{attribute 'GeneratedUsingTerminal: EL3201-0030-0022'}
{attribute addProperty BoxType "EL3201-0030-0022"}
{attribute addProperty Id "RTDAT %I*AI_Standard_Channel_4A3944819WcStateAT %I*WcState_9091E0EB2InfoDataAT %I*InfoData_94A18F5E2"}
{attribute addProperty CRC "3460650235"}
{attribute addProperty Size "13"}
TYPE EL3201_CE4554FB EXTENDS EtcSlaveTerminalBase_947E5A46 :
STRUCT
	{attribute addProperty Name "RTD"}
	RTD : AI_Standard_Channel_4A394481;
	{attribute addProperty Name "WcState"}
	WcState : WcState_9091E0EB;
	{attribute addProperty Name "InfoData"}
	InfoData : InfoData_94A18F5E;
END_STRUCT
END_TYPE

(* stored: Version 1.2.0.0, ProductVersion 3.1.4024.9
   DUT EL3201_CE4554FB: Id {fbf2789c-9caa-4dd7-bdbb-0410248806fb} *)
